// TIA Portal V17 export
// export: Created 2024-06-14T09:53:07.7504734Z, ExportSetting WithDefaults, DisplayName Totally Integrated Automation Portal, DisplayVersion V17, DisplayName TIA Portal Openness, DisplayVersion V17, DisplayName TIA Portal Version Control Interface, DisplayVersion V17, DisplayName Simotion SCOUT TIA, DisplayVersion 5.4.3.0, DisplayName SINAMICS Startdrive Advanced, DisplayVersion V17 SP1 Update 1, DisplayName SINAMICS Startdrive G110M, G120, G120C, G120D, G120P, G115D, DisplayVersion V17 SP1 Update 1, DisplayName SINAMICS Startdrive G130, G150, S120, S150, SINAMICS MV, S210, DisplayVersion V17 SP1 Update 1, DisplayName STEP 7 Professional, DisplayVersion V17, DisplayName STEP 7 Safety, DisplayVersion V17, DisplayName WinCC Professional, DisplayVersion V17
FUNCTION "CHECK_SCALE" : Void   // FC2, LAD
{ S7_Optimized_Access := 'TRUE' }
VERSION : 0.1
// stored: AutoNumber true, IsIECCheckEnabled false, SetENOAutomatically false, UDAEnableTagReadback false
   VAR_TEMP
      cycle_start : Bool;
      temp : Int;
   END_VAR
BEGIN

REGION Network 1
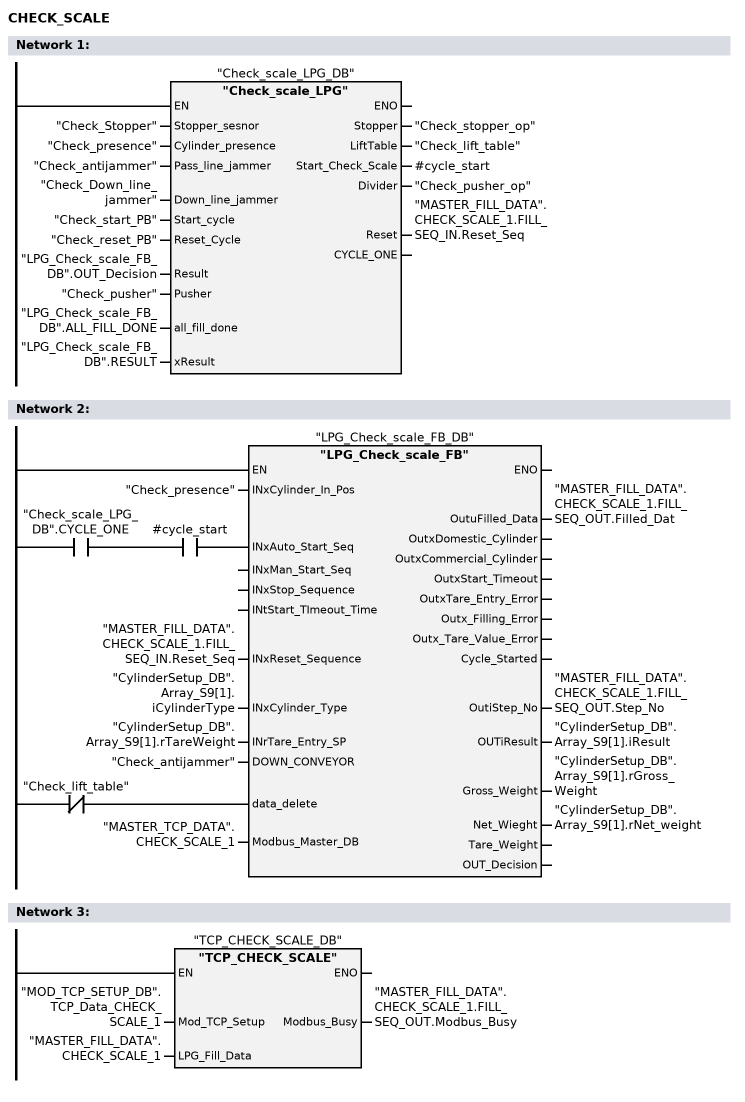
   RUNG wire#powerrail
      "Check_scale_LPG_DB"(Stopper_sesnor := "Check_Stopper", Cylinder_presence := "Check_presence", Pass_line_jammer := "Check_antijammer", Down_line_jammer := "Check_Down_line_jammer", Start_cycle := "Check_start_PB", Reset_Cycle := "Check_reset_PB", Result := "LPG_Check_scale_FB_DB".OUT_Decision, Pusher := "Check_pusher", all_fill_done := "LPG_Check_scale_FB_DB".ALL_FILL_DONE, xResult := "LPG_Check_scale_FB_DB".RESULT, Stopper => "Check_stopper_op", LiftTable => "Check_lift_table", Start_Check_Scale => #cycle_start, Divider => "Check_pusher_op", Reset => "MASTER_FILL_DATA".CHECK_SCALE_1.FILL_SEQ_IN.Reset_Seq, CYCLE_ONE =>)
   END_RUNG
   // the same network as SCL:
   "Check_scale_LPG_DB"(Stopper_sesnor := "Check_Stopper",   // "Check_scale_LPG"
                        Cylinder_presence := "Check_presence",
                        Pass_line_jammer := "Check_antijammer",
                        Down_line_jammer := "Check_Down_line_jammer",
                        Start_cycle := "Check_start_PB",
                        Reset_Cycle := "Check_reset_PB",
                        Result := "LPG_Check_scale_FB_DB".OUT_Decision,
                        Pusher := "Check_pusher",
                        all_fill_done := "LPG_Check_scale_FB_DB".ALL_FILL_DONE,
                        xResult := "LPG_Check_scale_FB_DB".RESULT,
                        Stopper => "Check_stopper_op",
                        LiftTable => "Check_lift_table",
                        Start_Check_Scale => #cycle_start,
                        Divider => "Check_pusher_op",
                        Reset => "MASTER_FILL_DATA".CHECK_SCALE_1.FILL_SEQ_IN.Reset_Seq);
END_REGION

REGION Network 2
   RUNG wire#powerrail
      "LPG_Check_scale_FB_DB"(INxAuto_Start_Seq := wire#w1, data_delete := wire#w2, INxCylinder_In_Pos := "Check_presence", INxMan_Start_Seq :=, INxStop_Sequence :=, INtStart_TImeout_Time :=, INxReset_Sequence := "MASTER_FILL_DATA".CHECK_SCALE_1.FILL_SEQ_IN.Reset_Seq, INxCylinder_Type := "CylinderSetup_DB".Array_S9[1].iCylinderType, INrTare_Entry_SP := "CylinderSetup_DB".Array_S9[1].rTareWeight, DOWN_CONVEYOR := "Check_antijammer", Modbus_Master_DB := "MASTER_TCP_DATA".CHECK_SCALE_1, OutuFilled_Data => "MASTER_FILL_DATA".CHECK_SCALE_1.FILL_SEQ_OUT.Filled_Dat, OutxDomestic_Cylinder =>, OutxCommercial_Cylinder =>, OutxStart_Timeout =>, OutxTare_Entry_Error =>, Outx_Filling_Error =>, Outx_Tare_Value_Error =>, Cycle_Started =>, OutiStep_No => "MASTER_FILL_DATA".CHECK_SCALE_1.FILL_SEQ_OUT.Step_No, OUTiResult => "CylinderSetup_DB".Array_S9[1].iResult, Gross_Weight => "CylinderSetup_DB".Array_S9[1].rGross_Weight, Net_Wieght => "CylinderSetup_DB".Array_S9[1].rNet_weight, Tare_Weight =>, OUT_Decision =>)
   END_RUNG
   RUNG wire#powerrail
      Contact( "Check_scale_LPG_DB".CYCLE_ONE )
      Contact( #cycle_start )
   END_RUNG wire#w1
   RUNG wire#powerrail
      I_Contact( "Check_lift_table" )
   END_RUNG wire#w2
   // the same network as SCL:
   "LPG_Check_scale_FB_DB"(INxCylinder_In_Pos := "Check_presence",   // "LPG_Check_scale_FB"
                           INxAuto_Start_Seq := "Check_scale_LPG_DB".CYCLE_ONE AND #cycle_start,
                           INxReset_Sequence := "MASTER_FILL_DATA".CHECK_SCALE_1.FILL_SEQ_IN.Reset_Seq,
                           INxCylinder_Type := "CylinderSetup_DB".Array_S9[1].iCylinderType,
                           INrTare_Entry_SP := "CylinderSetup_DB".Array_S9[1].rTareWeight,
                           DOWN_CONVEYOR := "Check_antijammer",
                           data_delete := NOT "Check_lift_table",
                           Modbus_Master_DB := "MASTER_TCP_DATA".CHECK_SCALE_1,
                           OutuFilled_Data => "MASTER_FILL_DATA".CHECK_SCALE_1.FILL_SEQ_OUT.Filled_Dat,
                           OutiStep_No => "MASTER_FILL_DATA".CHECK_SCALE_1.FILL_SEQ_OUT.Step_No,
                           OUTiResult => "CylinderSetup_DB".Array_S9[1].iResult,
                           Gross_Weight => "CylinderSetup_DB".Array_S9[1].rGross_Weight,
                           Net_Wieght => "CylinderSetup_DB".Array_S9[1].rNet_weight);
END_REGION

REGION Network 3
   RUNG wire#powerrail
      "TCP_CHECK_SCALE_DB"(Mod_TCP_Setup := "MOD_TCP_SETUP_DB".TCP_Data_CHECK_SCALE_1, LPG_Fill_Data := "MASTER_FILL_DATA".CHECK_SCALE_1, Modbus_Busy => "MASTER_FILL_DATA".CHECK_SCALE_1.FILL_SEQ_OUT.Modbus_Busy)
   END_RUNG
   // the same network as SCL:
   "TCP_CHECK_SCALE_DB"(Mod_TCP_Setup := "MOD_TCP_SETUP_DB".TCP_Data_CHECK_SCALE_1,   // "TCP_CHECK_SCALE"
                        LPG_Fill_Data := "MASTER_FILL_DATA".CHECK_SCALE_1,
                        Modbus_Busy => "MASTER_FILL_DATA".CHECK_SCALE_1.FILL_SEQ_OUT.Modbus_Busy);
END_REGION
END_FUNCTION
